// TIA Portal V17 export
// export: Created 2025-03-20T13:42:25.0446478Z, ExportSetting WithDefaults, DisplayName Totally Integrated Automation Portal, DisplayVersion V17 Update 8, DisplayName TIA Portal Openness, DisplayVersion V17 Update 8, DisplayName TIA Portal Version Control Interface, DisplayVersion V17, DisplayName SINAMICS Startdrive Advanced, DisplayVersion V17 SP2, DisplayName SINAMICS Startdrive G110M, G120, G120C, G120D, G120P, G115D, DisplayVersion V17 SP2, DisplayName SINAMICS Startdrive G130, G150, S120, S150, SINAMICS MV, S210, DisplayVersion V17 SP2, DisplayName STEP 7 Professional, DisplayVersion V17 Update 8, DisplayName SINUMERIK ONE STEP 7 Toolbox, DisplayVersion V17 Update 12, DisplayName SINUMERIK 840D sl STEP 7 Toolbox, DisplayVersion V17 Update 12, DisplayName STEP 7 Safety, DisplayVersion V17 Update 6, DisplayName WinCC Advanced, DisplayVersion V17 Update 8
FUNCTION_BLOCK "FB22301_SOLENOID_VALVE"   // FB22301, LAD
TITLE = FB22301 HOPPER FEED
{ S7_Optimized_Access := 'FALSE' }
VERSION : 0.1
// stored: AutoNumber false, IsIECCheckEnabled false, SetENOAutomatically false, UDAEnableTagReadback false
   VAR_INPUT
      iCONTROL_ON_DELAYED : Bool;
      iPNEUMATIC_FEEDBACK_ON : Bool;
      iMANUAL_START_REQUEST : Bool;
      iAUTO_START_REQUEST : Bool;
      iMANUAL_STOP_REQUEST : Bool;
      iAUTO_STOP_REQUEST : Bool;
   END_VAR
   VAR_OUTPUT
      oSYSTEM_ON : Bool;
   END_VAR
   VAR DB_SPECIFIC
      "DATA STANDARD" { S7_SetPoint := 'True'} : "GENERAL_DATA_START_STOP";
      "HMI STANDARD" { S7_SetPoint := 'True'} : "HMI_DATA_START_STOP";
   END_VAR
   VAR_TEMP
      DB_NUMBER : DInt;
   END_VAR
   VAR_TEMP   // added for the SCL form of the ladder/FBD networks
      _w1 : Bool;
   END_VAR
BEGIN

NETWORK
TITLE = READ INSTANCE DB NUMBER
      L     DINO;
      +     10#800000;
      T     #DB_NUMBER;

REGION Network 2: GENERAL CONDITIONS / Start General Conditions
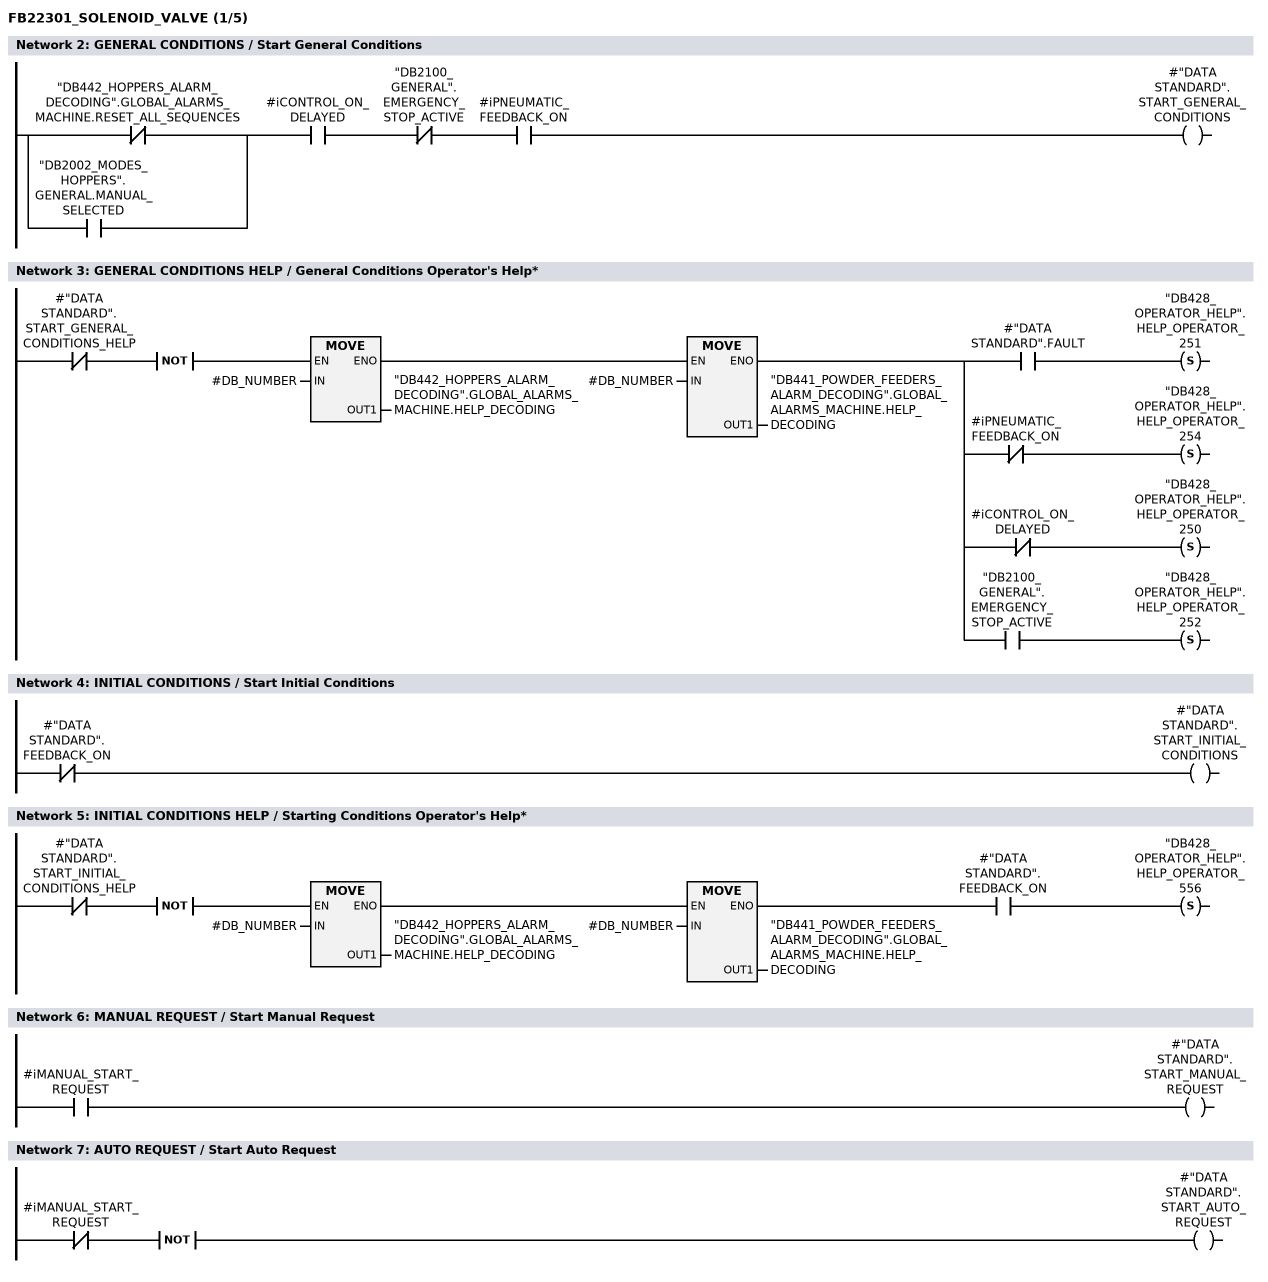
   RUNG wire#powerrail
      I_Contact( "DB442_HOPPERS_ALARM_DECODING".GLOBAL_ALARMS_MACHINE.RESET_ALL_SEQUENCES )
      wire#w1
      Contact( #iCONTROL_ON_DELAYED )
      I_Contact( "DB2100_GENERAL".EMERGENCY_STOP_ACTIVE )
      Contact( #iPNEUMATIC_FEEDBACK_ON )
      Coil( #"DATA STANDARD".START_GENERAL_CONDITIONS )
   END_RUNG
   RUNG wire#powerrail
      Contact( "DB2002_MODES_HOPPERS".GENERAL.MANUAL_SELECTED )
   END_RUNG wire#w1
   // the same network as SCL:
   #"DATA STANDARD".START_GENERAL_CONDITIONS := (NOT "DB442_HOPPERS_ALARM_DECODING".GLOBAL_ALARMS_MACHINE.RESET_ALL_SEQUENCES OR "DB2002_MODES_HOPPERS".GENERAL.MANUAL_SELECTED) AND #iCONTROL_ON_DELAYED AND NOT "DB2100_GENERAL".EMERGENCY_STOP_ACTIVE AND #iPNEUMATIC_FEEDBACK_ON;
END_REGION

REGION Network 3: GENERAL CONDITIONS HELP / General Conditions Operator's Help*
   RUNG wire#powerrail
      I_Contact( #"DATA STANDARD".START_GENERAL_CONDITIONS_HELP )
      Not()
      Move(in := #DB_NUMBER, out1 => "DB442_HOPPERS_ALARM_DECODING".GLOBAL_ALARMS_MACHINE.HELP_DECODING)
      Move(in := #DB_NUMBER, out1 => "DB441_POWDER_FEEDERS_ALARM_DECODING".GLOBAL_ALARMS_MACHINE.HELP_DECODING)
      wire#w1
      Contact( #"DATA STANDARD".FAULT )
      S_Coil( "DB428_OPERATOR_HELP".HELP_OPERATOR_251 )
   END_RUNG
   RUNG wire#w1
      I_Contact( #iPNEUMATIC_FEEDBACK_ON )
      S_Coil( "DB428_OPERATOR_HELP".HELP_OPERATOR_254 )
   END_RUNG
   RUNG wire#w1
      I_Contact( #iCONTROL_ON_DELAYED )
      S_Coil( "DB428_OPERATOR_HELP".HELP_OPERATOR_250 )
   END_RUNG
   RUNG wire#w1
      Contact( "DB2100_GENERAL".EMERGENCY_STOP_ACTIVE )
      S_Coil( "DB428_OPERATOR_HELP".HELP_OPERATOR_252 )
   END_RUNG
   // the same network as SCL:
   #_w1 := NOT (NOT #"DATA STANDARD".START_GENERAL_CONDITIONS_HELP);
   IF #_w1 THEN
       "DB442_HOPPERS_ALARM_DECODING".GLOBAL_ALARMS_MACHINE.HELP_DECODING := #DB_NUMBER;
       "DB441_POWDER_FEEDERS_ALARM_DECODING".GLOBAL_ALARMS_MACHINE.HELP_DECODING := #DB_NUMBER;
   END_IF;
   IF #_w1 AND #"DATA STANDARD".FAULT THEN "DB428_OPERATOR_HELP".HELP_OPERATOR_251 := TRUE; END_IF;
   IF #_w1 AND NOT #iPNEUMATIC_FEEDBACK_ON THEN "DB428_OPERATOR_HELP".HELP_OPERATOR_254 := TRUE; END_IF;
   IF #_w1 AND NOT #iCONTROL_ON_DELAYED THEN "DB428_OPERATOR_HELP".HELP_OPERATOR_250 := TRUE; END_IF;
   IF #_w1 AND "DB2100_GENERAL".EMERGENCY_STOP_ACTIVE THEN
       "DB428_OPERATOR_HELP".HELP_OPERATOR_252 := TRUE;
   END_IF;
END_REGION

REGION Network 4: INITIAL CONDITIONS / Start Initial Conditions
   RUNG wire#powerrail
      I_Contact( #"DATA STANDARD".FEEDBACK_ON )
      Coil( #"DATA STANDARD".START_INITIAL_CONDITIONS )
   END_RUNG
   // the same network as SCL:
   #"DATA STANDARD".START_INITIAL_CONDITIONS := NOT #"DATA STANDARD".FEEDBACK_ON;
END_REGION

REGION Network 5: INITIAL CONDITIONS HELP / Starting Conditions Operator's Help*
   RUNG wire#powerrail
      I_Contact( #"DATA STANDARD".START_INITIAL_CONDITIONS_HELP )
      Not()
      Move(in := #DB_NUMBER, out1 => "DB442_HOPPERS_ALARM_DECODING".GLOBAL_ALARMS_MACHINE.HELP_DECODING)
      Move(in := #DB_NUMBER, out1 => "DB441_POWDER_FEEDERS_ALARM_DECODING".GLOBAL_ALARMS_MACHINE.HELP_DECODING)
      Contact( #"DATA STANDARD".FEEDBACK_ON )
      S_Coil( "DB428_OPERATOR_HELP".HELP_OPERATOR_556 )
   END_RUNG
   // the same network as SCL:
   #_w1 := NOT (NOT #"DATA STANDARD".START_INITIAL_CONDITIONS_HELP);
   IF #_w1 THEN
       "DB442_HOPPERS_ALARM_DECODING".GLOBAL_ALARMS_MACHINE.HELP_DECODING := #DB_NUMBER;
       "DB441_POWDER_FEEDERS_ALARM_DECODING".GLOBAL_ALARMS_MACHINE.HELP_DECODING := #DB_NUMBER;
   END_IF;
   IF #_w1 AND #"DATA STANDARD".FEEDBACK_ON THEN "DB428_OPERATOR_HELP".HELP_OPERATOR_556 := TRUE; END_IF;
END_REGION

REGION Network 6: MANUAL REQUEST / Start Manual Request
   RUNG wire#powerrail
      Contact( #iMANUAL_START_REQUEST )
      Coil( #"DATA STANDARD".START_MANUAL_REQUEST )
   END_RUNG
   // the same network as SCL:
   #"DATA STANDARD".START_MANUAL_REQUEST := #iMANUAL_START_REQUEST;
END_REGION

REGION Network 7: AUTO REQUEST / Start Auto Request
   RUNG wire#powerrail
      I_Contact( #iMANUAL_START_REQUEST )
      Not()
      Coil( #"DATA STANDARD".START_AUTO_REQUEST )
   END_RUNG
   // the same network as SCL:
   #"DATA STANDARD".START_AUTO_REQUEST := NOT (NOT #iMANUAL_START_REQUEST);
END_REGION

REGION Network 8: GLOBAL REQUEST / Start Global Request
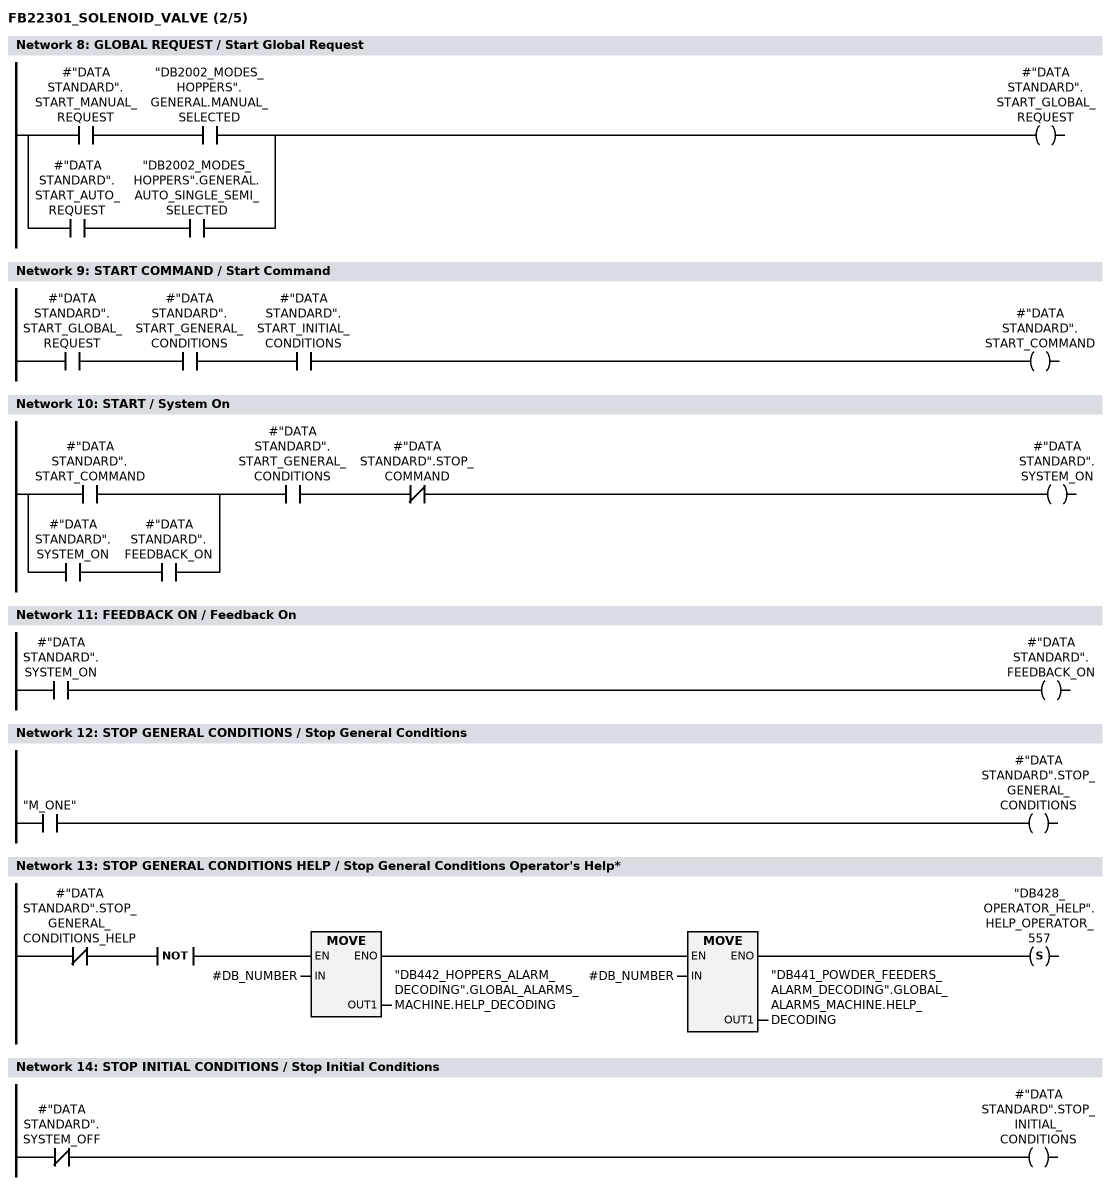
   RUNG wire#powerrail
      Contact( #"DATA STANDARD".START_MANUAL_REQUEST )
      Contact( "DB2002_MODES_HOPPERS".GENERAL.MANUAL_SELECTED )
      wire#w1
      Coil( #"DATA STANDARD".START_GLOBAL_REQUEST )
   END_RUNG
   RUNG wire#powerrail
      Contact( #"DATA STANDARD".START_AUTO_REQUEST )
      Contact( "DB2002_MODES_HOPPERS".GENERAL.AUTO_SINGLE_SEMI_SELECTED )
   END_RUNG wire#w1
   // the same network as SCL:
   #"DATA STANDARD".START_GLOBAL_REQUEST := (#"DATA STANDARD".START_MANUAL_REQUEST AND "DB2002_MODES_HOPPERS".GENERAL.MANUAL_SELECTED) OR (#"DATA STANDARD".START_AUTO_REQUEST AND "DB2002_MODES_HOPPERS".GENERAL.AUTO_SINGLE_SEMI_SELECTED);
END_REGION

REGION Network 9: START COMMAND / Start Command
   RUNG wire#powerrail
      Contact( #"DATA STANDARD".START_GLOBAL_REQUEST )
      Contact( #"DATA STANDARD".START_GENERAL_CONDITIONS )
      Contact( #"DATA STANDARD".START_INITIAL_CONDITIONS )
      Coil( #"DATA STANDARD".START_COMMAND )
   END_RUNG
   // the same network as SCL:
   #"DATA STANDARD".START_COMMAND := #"DATA STANDARD".START_GLOBAL_REQUEST AND #"DATA STANDARD".START_GENERAL_CONDITIONS AND #"DATA STANDARD".START_INITIAL_CONDITIONS;
END_REGION

REGION Network 10: START / System On
   RUNG wire#powerrail
      Contact( #"DATA STANDARD".START_COMMAND )
      wire#w1
      Contact( #"DATA STANDARD".START_GENERAL_CONDITIONS )
      I_Contact( #"DATA STANDARD".STOP_COMMAND )
      Coil( #"DATA STANDARD".SYSTEM_ON )
   END_RUNG
   RUNG wire#powerrail
      Contact( #"DATA STANDARD".SYSTEM_ON )
      Contact( #"DATA STANDARD".FEEDBACK_ON )
   END_RUNG wire#w1
   // the same network as SCL:
   #"DATA STANDARD".SYSTEM_ON := (#"DATA STANDARD".START_COMMAND OR (#"DATA STANDARD".SYSTEM_ON AND #"DATA STANDARD".FEEDBACK_ON)) AND #"DATA STANDARD".START_GENERAL_CONDITIONS AND NOT #"DATA STANDARD".STOP_COMMAND;
END_REGION

REGION Network 11: FEEDBACK ON / Feedback On
   RUNG wire#powerrail
      Contact( #"DATA STANDARD".SYSTEM_ON )
      Coil( #"DATA STANDARD".FEEDBACK_ON )
   END_RUNG
   // the same network as SCL:
   #"DATA STANDARD".FEEDBACK_ON := #"DATA STANDARD".SYSTEM_ON;
END_REGION

REGION Network 12: STOP GENERAL CONDITIONS / Stop General Conditions
   RUNG wire#powerrail
      Contact( "M_ONE" )
      Coil( #"DATA STANDARD".STOP_GENERAL_CONDITIONS )
   END_RUNG
   // the same network as SCL:
   #"DATA STANDARD".STOP_GENERAL_CONDITIONS := "M_ONE";
END_REGION

REGION Network 13: STOP GENERAL CONDITIONS HELP / Stop General Conditions Operator's Help*
   RUNG wire#powerrail
      I_Contact( #"DATA STANDARD".STOP_GENERAL_CONDITIONS_HELP )
      Not()
      Move(in := #DB_NUMBER, out1 => "DB442_HOPPERS_ALARM_DECODING".GLOBAL_ALARMS_MACHINE.HELP_DECODING)
      Move(in := #DB_NUMBER, out1 => "DB441_POWDER_FEEDERS_ALARM_DECODING".GLOBAL_ALARMS_MACHINE.HELP_DECODING)
      S_Coil( "DB428_OPERATOR_HELP".HELP_OPERATOR_557 )
   END_RUNG
   // the same network as SCL:
   IF NOT (NOT #"DATA STANDARD".STOP_GENERAL_CONDITIONS_HELP) THEN
       "DB442_HOPPERS_ALARM_DECODING".GLOBAL_ALARMS_MACHINE.HELP_DECODING := #DB_NUMBER;
       "DB441_POWDER_FEEDERS_ALARM_DECODING".GLOBAL_ALARMS_MACHINE.HELP_DECODING := #DB_NUMBER;
       "DB428_OPERATOR_HELP".HELP_OPERATOR_557 := TRUE;
   END_IF;
END_REGION

REGION Network 14: STOP INITIAL CONDITIONS / Stop Initial Conditions
   RUNG wire#powerrail
      I_Contact( #"DATA STANDARD".SYSTEM_OFF )
      Coil( #"DATA STANDARD".STOP_INITIAL_CONDITIONS )
   END_RUNG
   // the same network as SCL:
   #"DATA STANDARD".STOP_INITIAL_CONDITIONS := NOT #"DATA STANDARD".SYSTEM_OFF;
END_REGION

REGION Network 15: STOP INITIAL CONDITIONS HELP / Stop Inital Conditions Operator's Help*
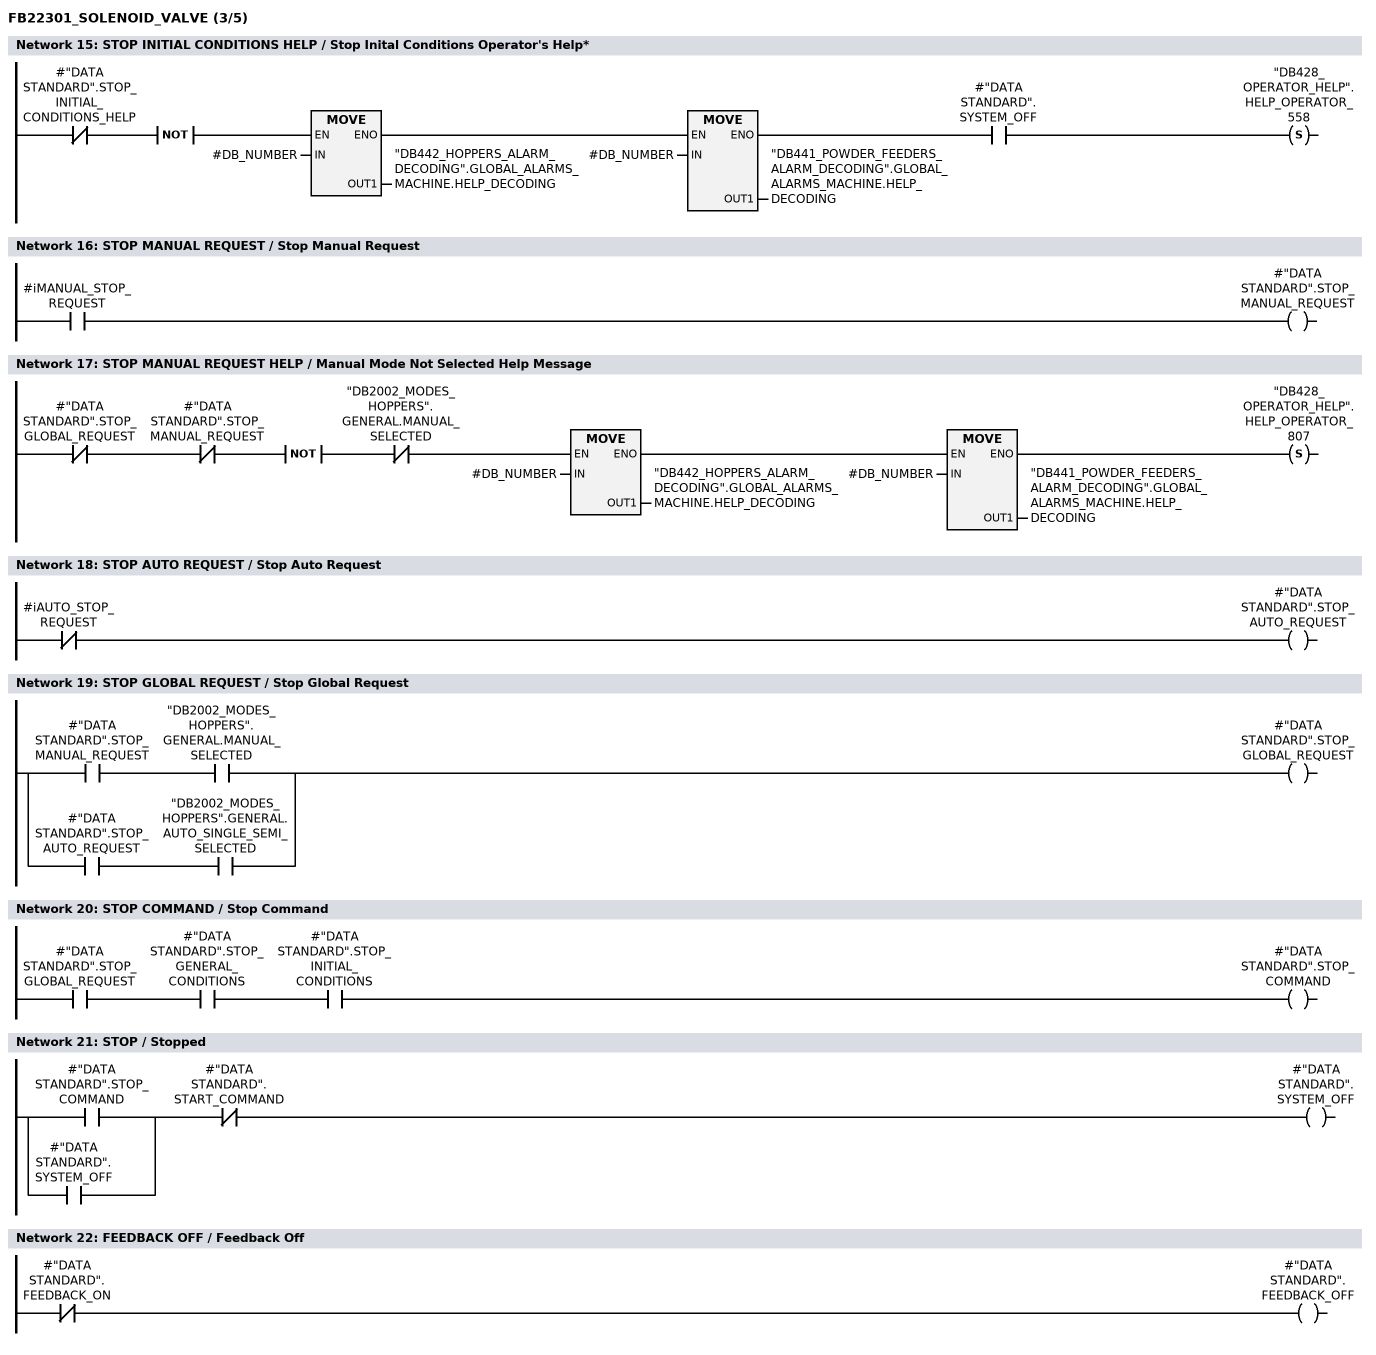
   RUNG wire#powerrail
      I_Contact( #"DATA STANDARD".STOP_INITIAL_CONDITIONS_HELP )
      Not()
      Move(in := #DB_NUMBER, out1 => "DB442_HOPPERS_ALARM_DECODING".GLOBAL_ALARMS_MACHINE.HELP_DECODING)
      Move(in := #DB_NUMBER, out1 => "DB441_POWDER_FEEDERS_ALARM_DECODING".GLOBAL_ALARMS_MACHINE.HELP_DECODING)
      Contact( #"DATA STANDARD".SYSTEM_OFF )
      S_Coil( "DB428_OPERATOR_HELP".HELP_OPERATOR_558 )
   END_RUNG
   // the same network as SCL:
   #_w1 := NOT (NOT #"DATA STANDARD".STOP_INITIAL_CONDITIONS_HELP);
   IF #_w1 THEN
       "DB442_HOPPERS_ALARM_DECODING".GLOBAL_ALARMS_MACHINE.HELP_DECODING := #DB_NUMBER;
       "DB441_POWDER_FEEDERS_ALARM_DECODING".GLOBAL_ALARMS_MACHINE.HELP_DECODING := #DB_NUMBER;
   END_IF;
   IF #_w1 AND #"DATA STANDARD".SYSTEM_OFF THEN "DB428_OPERATOR_HELP".HELP_OPERATOR_558 := TRUE; END_IF;
END_REGION

REGION Network 16: STOP MANUAL REQUEST / Stop Manual Request
   RUNG wire#powerrail
      Contact( #iMANUAL_STOP_REQUEST )
      Coil( #"DATA STANDARD".STOP_MANUAL_REQUEST )
   END_RUNG
   // the same network as SCL:
   #"DATA STANDARD".STOP_MANUAL_REQUEST := #iMANUAL_STOP_REQUEST;
END_REGION

REGION Network 17: STOP MANUAL REQUEST HELP / Manual Mode Not Selected Help Message
   RUNG wire#powerrail
      I_Contact( #"DATA STANDARD".STOP_GLOBAL_REQUEST )
      I_Contact( #"DATA STANDARD".STOP_MANUAL_REQUEST )
      Not()
      I_Contact( "DB2002_MODES_HOPPERS".GENERAL.MANUAL_SELECTED )
      Move(in := #DB_NUMBER, out1 => "DB442_HOPPERS_ALARM_DECODING".GLOBAL_ALARMS_MACHINE.HELP_DECODING)
      Move(in := #DB_NUMBER, out1 => "DB441_POWDER_FEEDERS_ALARM_DECODING".GLOBAL_ALARMS_MACHINE.HELP_DECODING)
      S_Coil( "DB428_OPERATOR_HELP".HELP_OPERATOR_807 )
   END_RUNG
   // the same network as SCL:
   IF NOT (NOT #"DATA STANDARD".STOP_GLOBAL_REQUEST AND NOT #"DATA STANDARD".STOP_MANUAL_REQUEST) AND NOT "DB2002_MODES_HOPPERS".GENERAL.MANUAL_SELECTED THEN
       "DB442_HOPPERS_ALARM_DECODING".GLOBAL_ALARMS_MACHINE.HELP_DECODING := #DB_NUMBER;
       "DB441_POWDER_FEEDERS_ALARM_DECODING".GLOBAL_ALARMS_MACHINE.HELP_DECODING := #DB_NUMBER;
       "DB428_OPERATOR_HELP".HELP_OPERATOR_807 := TRUE;
   END_IF;
END_REGION

REGION Network 18: STOP AUTO REQUEST / Stop Auto Request
   RUNG wire#powerrail
      I_Contact( #iAUTO_STOP_REQUEST )
      Coil( #"DATA STANDARD".STOP_AUTO_REQUEST )
   END_RUNG
   // the same network as SCL:
   #"DATA STANDARD".STOP_AUTO_REQUEST := NOT #iAUTO_STOP_REQUEST;
END_REGION

REGION Network 19: STOP GLOBAL REQUEST / Stop Global Request
   RUNG wire#powerrail
      Contact( #"DATA STANDARD".STOP_MANUAL_REQUEST )
      Contact( "DB2002_MODES_HOPPERS".GENERAL.MANUAL_SELECTED )
      wire#w1
      Coil( #"DATA STANDARD".STOP_GLOBAL_REQUEST )
   END_RUNG
   RUNG wire#powerrail
      Contact( #"DATA STANDARD".STOP_AUTO_REQUEST )
      Contact( "DB2002_MODES_HOPPERS".GENERAL.AUTO_SINGLE_SEMI_SELECTED )
   END_RUNG wire#w1
   // the same network as SCL:
   #"DATA STANDARD".STOP_GLOBAL_REQUEST := (#"DATA STANDARD".STOP_MANUAL_REQUEST AND "DB2002_MODES_HOPPERS".GENERAL.MANUAL_SELECTED) OR (#"DATA STANDARD".STOP_AUTO_REQUEST AND "DB2002_MODES_HOPPERS".GENERAL.AUTO_SINGLE_SEMI_SELECTED);
END_REGION

REGION Network 20: STOP COMMAND / Stop Command
   RUNG wire#powerrail
      Contact( #"DATA STANDARD".STOP_GLOBAL_REQUEST )
      Contact( #"DATA STANDARD".STOP_GENERAL_CONDITIONS )
      Contact( #"DATA STANDARD".STOP_INITIAL_CONDITIONS )
      Coil( #"DATA STANDARD".STOP_COMMAND )
   END_RUNG
   // the same network as SCL:
   #"DATA STANDARD".STOP_COMMAND := #"DATA STANDARD".STOP_GLOBAL_REQUEST AND #"DATA STANDARD".STOP_GENERAL_CONDITIONS AND #"DATA STANDARD".STOP_INITIAL_CONDITIONS;
END_REGION

REGION Network 21: STOP / Stopped
   RUNG wire#powerrail
      Contact( #"DATA STANDARD".STOP_COMMAND )
      wire#w1
      I_Contact( #"DATA STANDARD".START_COMMAND )
      Coil( #"DATA STANDARD".SYSTEM_OFF )
   END_RUNG
   RUNG wire#powerrail
      Contact( #"DATA STANDARD".SYSTEM_OFF )
   END_RUNG wire#w1
   // the same network as SCL:
   #"DATA STANDARD".SYSTEM_OFF := (#"DATA STANDARD".STOP_COMMAND OR #"DATA STANDARD".SYSTEM_OFF) AND NOT #"DATA STANDARD".START_COMMAND;
END_REGION

REGION Network 22: FEEDBACK OFF / Feedback Off
   RUNG wire#powerrail
      I_Contact( #"DATA STANDARD".FEEDBACK_ON )
      Coil( #"DATA STANDARD".FEEDBACK_OFF )
   END_RUNG
   // the same network as SCL:
   #"DATA STANDARD".FEEDBACK_OFF := NOT #"DATA STANDARD".FEEDBACK_ON;
END_REGION

REGION Network 23: RESET / Laser System Fault
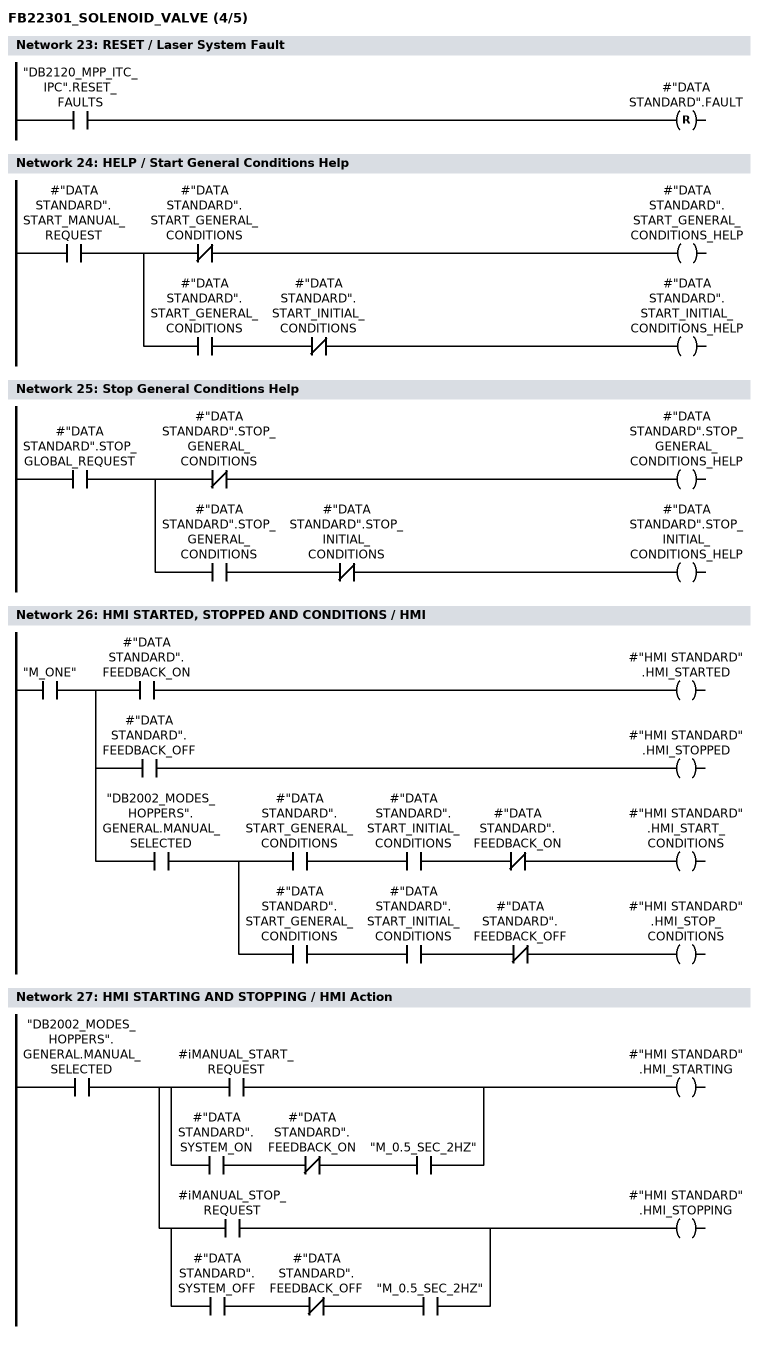
   RUNG wire#powerrail
      Contact( "DB2120_MPP_ITC_IPC".RESET_FAULTS )
      R_Coil( #"DATA STANDARD".FAULT )
   END_RUNG
   // the same network as SCL:
   IF "DB2120_MPP_ITC_IPC".RESET_FAULTS THEN #"DATA STANDARD".FAULT := FALSE; END_IF;
END_REGION

REGION Network 24: HELP / Start General Conditions Help
   RUNG wire#powerrail
      Contact( #"DATA STANDARD".START_MANUAL_REQUEST )
      wire#w1
      I_Contact( #"DATA STANDARD".START_GENERAL_CONDITIONS )
      Coil( #"DATA STANDARD".START_GENERAL_CONDITIONS_HELP )
   END_RUNG
   RUNG wire#w1
      Contact( #"DATA STANDARD".START_GENERAL_CONDITIONS )
      I_Contact( #"DATA STANDARD".START_INITIAL_CONDITIONS )
      Coil( #"DATA STANDARD".START_INITIAL_CONDITIONS_HELP )
   END_RUNG
   // the same network as SCL:
   #"DATA STANDARD".START_GENERAL_CONDITIONS_HELP := #"DATA STANDARD".START_MANUAL_REQUEST AND NOT #"DATA STANDARD".START_GENERAL_CONDITIONS;
   #"DATA STANDARD".START_INITIAL_CONDITIONS_HELP := #"DATA STANDARD".START_MANUAL_REQUEST AND #"DATA STANDARD".START_GENERAL_CONDITIONS AND NOT #"DATA STANDARD".START_INITIAL_CONDITIONS;
END_REGION

REGION Network 25: Stop General Conditions Help
   RUNG wire#powerrail
      Contact( #"DATA STANDARD".STOP_GLOBAL_REQUEST )
      wire#w1
      I_Contact( #"DATA STANDARD".STOP_GENERAL_CONDITIONS )
      Coil( #"DATA STANDARD".STOP_GENERAL_CONDITIONS_HELP )
   END_RUNG
   RUNG wire#w1
      Contact( #"DATA STANDARD".STOP_GENERAL_CONDITIONS )
      I_Contact( #"DATA STANDARD".STOP_INITIAL_CONDITIONS )
      Coil( #"DATA STANDARD".STOP_INITIAL_CONDITIONS_HELP )
   END_RUNG
   // the same network as SCL:
   #"DATA STANDARD".STOP_GENERAL_CONDITIONS_HELP := #"DATA STANDARD".STOP_GLOBAL_REQUEST AND NOT #"DATA STANDARD".STOP_GENERAL_CONDITIONS;
   #"DATA STANDARD".STOP_INITIAL_CONDITIONS_HELP := #"DATA STANDARD".STOP_GLOBAL_REQUEST AND #"DATA STANDARD".STOP_GENERAL_CONDITIONS AND NOT #"DATA STANDARD".STOP_INITIAL_CONDITIONS;
END_REGION

REGION Network 26: HMI STARTED, STOPPED AND CONDITIONS / HMI
   RUNG wire#powerrail
      Contact( "M_ONE" )
      wire#w1
      Contact( #"DATA STANDARD".FEEDBACK_ON )
      Coil( #"HMI STANDARD".HMI_STARTED )
   END_RUNG
   RUNG wire#w1
      Contact( #"DATA STANDARD".FEEDBACK_OFF )
      Coil( #"HMI STANDARD".HMI_STOPPED )
   END_RUNG
   RUNG wire#w1
      Contact( "DB2002_MODES_HOPPERS".GENERAL.MANUAL_SELECTED )
      wire#w2
      Contact( #"DATA STANDARD".START_GENERAL_CONDITIONS )
      Contact( #"DATA STANDARD".START_INITIAL_CONDITIONS )
      I_Contact( #"DATA STANDARD".FEEDBACK_ON )
      Coil( #"HMI STANDARD".HMI_START_CONDITIONS )
   END_RUNG
   RUNG wire#w2
      Contact( #"DATA STANDARD".START_GENERAL_CONDITIONS )
      Contact( #"DATA STANDARD".START_INITIAL_CONDITIONS )
      I_Contact( #"DATA STANDARD".FEEDBACK_OFF )
      Coil( #"HMI STANDARD".HMI_STOP_CONDITIONS )
   END_RUNG
   // the same network as SCL:
   #"HMI STANDARD".HMI_STARTED := "M_ONE" AND #"DATA STANDARD".FEEDBACK_ON;
   #"HMI STANDARD".HMI_STOPPED := "M_ONE" AND #"DATA STANDARD".FEEDBACK_OFF;
   #_w1 := "M_ONE" AND "DB2002_MODES_HOPPERS".GENERAL.MANUAL_SELECTED;
   #"HMI STANDARD".HMI_START_CONDITIONS := #_w1 AND #"DATA STANDARD".START_GENERAL_CONDITIONS AND #"DATA STANDARD".START_INITIAL_CONDITIONS AND NOT #"DATA STANDARD".FEEDBACK_ON;
   #"HMI STANDARD".HMI_STOP_CONDITIONS := #_w1 AND #"DATA STANDARD".START_GENERAL_CONDITIONS AND #"DATA STANDARD".START_INITIAL_CONDITIONS AND NOT #"DATA STANDARD".FEEDBACK_OFF;
END_REGION

REGION Network 27: HMI STARTING AND STOPPING / HMI Action
   RUNG wire#powerrail
      Contact( "DB2002_MODES_HOPPERS".GENERAL.MANUAL_SELECTED )
      wire#w1
      Contact( #iMANUAL_START_REQUEST )
      wire#w2
      Coil( #"HMI STANDARD".HMI_STARTING )
   END_RUNG
   RUNG wire#w1
      Contact( #"DATA STANDARD".SYSTEM_ON )
      I_Contact( #"DATA STANDARD".FEEDBACK_ON )
      Contact( "M_0.5_SEC_2HZ" )
   END_RUNG wire#w2
   RUNG wire#w1
      Contact( #iMANUAL_STOP_REQUEST )
      wire#w3
      Coil( #"HMI STANDARD".HMI_STOPPING )
   END_RUNG
   RUNG wire#w1
      Contact( #"DATA STANDARD".SYSTEM_OFF )
      I_Contact( #"DATA STANDARD".FEEDBACK_OFF )
      Contact( "M_0.5_SEC_2HZ" )
   END_RUNG wire#w3
   // the same network as SCL:
   #"HMI STANDARD".HMI_STARTING := "DB2002_MODES_HOPPERS".GENERAL.MANUAL_SELECTED AND (#iMANUAL_START_REQUEST OR (#"DATA STANDARD".SYSTEM_ON AND NOT #"DATA STANDARD".FEEDBACK_ON AND "M_0.5_SEC_2HZ"));
   #"HMI STANDARD".HMI_STOPPING := "DB2002_MODES_HOPPERS".GENERAL.MANUAL_SELECTED AND (#iMANUAL_STOP_REQUEST OR (#"DATA STANDARD".SYSTEM_OFF AND NOT #"DATA STANDARD".FEEDBACK_OFF AND "M_0.5_SEC_2HZ"));
END_REGION

REGION Network 28: OUTPUT / Output - Optic Blow
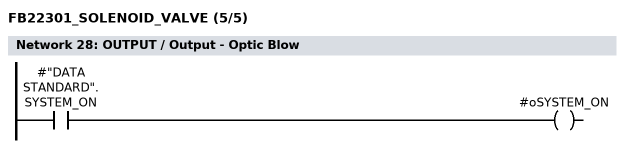
   RUNG wire#powerrail
      Contact( #"DATA STANDARD".SYSTEM_ON )
      Coil( #oSYSTEM_ON )
   END_RUNG
   // the same network as SCL:
   #oSYSTEM_ON := #"DATA STANDARD".SYSTEM_ON;
END_REGION
END_FUNCTION_BLOCK
